// TIA Portal V20 export
DATA_BLOCK "Trades_Calls"   // DB490
// stored: Access Published, MemoryReserve 100, Namespace CITI_Logic
   VAR
      Call : Array[1..5] of "CITI_Logic.zu_CallData";
   END_VAR
BEGIN
END_DATA_BLOCK
